FUNCTION F_Even : BOOL
VAR_INPUT
	uiNumber		: UINT;
END_VAR
VAR
END_VAR

F_Even := uiNumber MOD 2 = 0;

END_FUNCTION

(* stored: Version 1.1.0.1, ProductVersion 3.1.4024.13
   POU F_Even: Id {382c4f13-5c45-4d0f-8f4f-b79be49c4e37}, SpecialFunc None *)
